Fanuc KAREL source: kx00022.KL

PROGRAM KX00022
%NOLOCKGROUP
VAR
I:INTEGER;J:INTEGER;B:BOOLEAN
F : FILE
S : STRING[80]
P : XYZWPR
BA : ARRAY[4] OF BOOLEAN
BEGIN
--
--
BA[1]=TRUE
B=BA[1]
END KX00022
